{attribute 'GeneratedUsingTerminal: EP2816-0003-0016'}
{attribute addProperty BoxType "EP2816-0003-0016"}
{attribute addProperty Id "OutputAT %Q*ARRAY[0..7] OF BOOL8"}
{attribute addProperty CRC "1253840710"}
{attribute addProperty Size "8"}
TYPE DIG_Output_Channel_28AC1A9E :
STRUCT
	{attribute addProperty Name "Output"}
	Output AT %Q* : ARRAY[0..7] OF BOOL;
END_STRUCT
END_TYPE

(* stored: Version 1.2.0.0, ProductVersion 3.1.4024.9
   DUT DIG_Output_Channel_28AC1A9E: Id {7cf3aa51-3518-46c8-8b0a-1da7cbf30927} *)
